TEXTLIST TL_Mode
  0 = 'Tune'
  1 = 'Run'
   = ''
END_TEXTLIST

(* stored: Version 1.1.0.1, ProductVersion 3.1.4024.12
   TextList TL_Mode: Id {5713fa01-106c-4155-a89c-e267831ece75} *)
